{attribute 'GeneratedUsingTerminal: EQ1008-0002-0016'}
{attribute addProperty BoxType "EQ1008-0002-0016"}
{attribute addProperty Id "InputAT %I*BOOL1"}
{attribute addProperty CRC "2198356929"}
{attribute addProperty Size "1"}
TYPE Channel_830843C1 :
STRUCT
	{attribute addProperty Name "Input"}
	Input AT %I* : BOOL;
END_STRUCT
END_TYPE

(* stored: Version 1.2.0.0, ProductVersion 3.1.4024.9
   DUT Channel_830843C1: Id {c4882b63-ad37-44f5-867b-ad8b9124af7f} *)
